TYPE ST_BrakeParam :
STRUCT
	Deceleration 	: LREAL;
	Jerk 		: LREAL;
END_STRUCT
END_TYPE

(* stored: Version 1.1.0.1, ProductVersion 3.1.4024.9
   DUT ST_BrakeParam: Id {0473c4bf-df68-425f-92d6-46847dae84d4} *)
